GLOBALCONSTANTS AID_PG (* Picture graphic object attribute ids *)
  (* Standard: 61499-1; Description: Copyright (c) 2023 HR Agrartechnik GmbH This program and the accompanying materials are made available under the terms of the Eclipse Public License 2.0 which is available at https://www.eclipse.org/legal/epl-2.0/ SPDX-License-Identifier: EPL-2.0 *)
  (* Version 1.0, 2026-06-20, Franz Höpfinger, HR Agrartechnik GmbH *)
  PACKAGE isobus::UT::Q::const::AID;
  VAR_GLOBAL CONSTANT
    WIDTH : USINT := USINT#1; (* 1: AID_PG_WIDTH - Width in pixels. *)
    OPTIONS : USINT := USINT#2; (* 2: AID_PG_OPTIONS - Bitmask: Bit 0=Transparent, Bit 1=Flashing, Bit 2=Run-Length Encoded (RLE) *)
    TRANSPARENCY_COLOUR : USINT := USINT#3; (* 3: AID_PG_TRANSPARENCY_COLOUR *)
    ACTUAL_WIDTH : USINT := USINT#4; (* 4: AID_PG_ACTUAL_WIDTH (read-only) *)
    ACTUAL_HEIGHT : USINT := USINT#5; (* 5: AID_PG_ACTUAL_HEIGHT (read-only) *)
    FORMAT : USINT := USINT#6; (* 6: AID_PG_FORMAT (read-only) - Picture graphic type: 0 = Monochrome, 1 = 4-bit colour, 2 = 8-bit colour. *)
  END_VAR
END_GLOBALCONSTANTS
